{attribute 'linkalways'} 
{attribute 'no_explicit_call' := 'This FB is a CLASS and must be accessed using methods or properties'}
{attribute 'enable_dynamic_creation'}
FUNCTION_BLOCK AsyncCommand EXTENDS Disposable IMPLEMENTS I_AsyncCommand
VAR
	stateMachine : AsyncCommandStateMachine;
END_VAR

METHOD PUBLIC Abort
VAR_INPUT
END_VAR
stateMachine.Abort();
END_METHOD

PROPERTY PUBLIC Busy : BOOL
GET
IF stateMachine.IsAborted THEN
	RETURN;
END_IF

IF stateMachine.IsCompleted THEN
	RETURN;
END_IF

IF stateMachine.IsErrored THEN
	RETURN;
END_IF

IF stateMachine.IsIdle THEN
	RETURN;
END_IF

Busy := TRUE;
END_GET
END_PROPERTY

METHOD PUBLIC CyclicCall
VAR_INPUT
END_VAR
IF stateMachine.IsIdle THEN
	OnIdle();
END_IF

IF stateMachine.IsInitializing THEN
	OnInitializing(stateMachine);
END_IF

IF stateMachine.IsExecuting THEN
	OnExecuting(stateMachine);
END_IF

IF stateMachine.IsCompleting THEN
	OnCompleting(stateMachine);
END_IF

IF stateMachine.IsCompleted THEN
	OnCompleted();
END_IF

IF stateMachine.IsAborting THEN
	OnAborting(stateMachine);
END_IF

IF stateMachine.IsAborted THEN
	OnAborted();
END_IF

IF stateMachine.IsErrored THEN
	OnErrored();
END_IF
END_METHOD

PROPERTY PUBLIC Done : BOOL
GET
Done := stateMachine.IsCompleted;
END_GET
END_PROPERTY

PROPERTY PUBLIC Error : BOOL
GET
Error := stateMachine.IsErrored;
END_GET
END_PROPERTY

PROPERTY PUBLIC ErrorId : UDINT
GET
ErrorId := stateMachine.ErrorId;
END_GET
END_PROPERTY

METHOD PUBLIC Execute
VAR_INPUT
END_VAR
stateMachine.Execute();
END_METHOD

METHOD PROTECTED OnAborted
VAR_INPUT
END_VAR
END_METHOD

METHOD PROTECTED OnAborting
VAR_INPUT
	StateControl : I_AsyncCommandStateControl;
END_VAR
// default behaviour is to go to next state
// you can override this method to implement your own completing control code.
// just call StateControl.Next() when your code is completed.  

StateControl.Next();
END_METHOD

METHOD PROTECTED OnCompleted : BOOL
VAR_INPUT
END_VAR
END_METHOD

METHOD PROTECTED OnCompleting
VAR_INPUT
	StateControl : I_AsyncCommandStateControl;
END_VAR
// default behaviour is to go to next state
// you can override this method to implement your own completing control code.
// just call StateControl.Next() when your code is completed.  

StateControl.Next();
END_METHOD

METHOD PROTECTED OnErrored
VAR_INPUT
END_VAR
END_METHOD

METHOD PROTECTED OnExecuting
VAR_INPUT
	StateControl : I_AsyncCommandStateControl;
END_VAR
// default behaviour is to go to next state
// you can override this method to implement your own executing control code.
// just call StateControl.Next() when your code is completed.  

StateControl.Next();
END_METHOD

METHOD PROTECTED OnIdle
VAR_INPUT
END_VAR
END_METHOD

METHOD PROTECTED OnInitializing
VAR_INPUT
	StateControl : I_AsyncCommandStateControl;
END_VAR
// default behaviour is to go to next state
// you can override this method to implement your own initializing control code.
// just call StateControl.Next() when your code is completed.  

StateControl.Next();
END_METHOD

END_FUNCTION_BLOCK

(* stored: Version 1.1.0.1, ProductVersion 3.1.4024.12
   POU AsyncCommand: Id {c973928e-4f5b-09d1-33f2-08f2e9394838}, SpecialFunc None
   Folder Protected: Id {5a39a5d2-86a8-08f5-2eea-c36e6bea10ac}
   Method Abort: Id {7fe7ef70-8f92-07c8-094c-3e23fcd2f4b9}
   Property Busy: Id {41fde25d-7c78-0f8a-2bd6-3c43629fa217}
   Get Get: Id {50fe8db0-7c48-03a5-182b-c8bbcc843bb1}
   Method CyclicCall: Id {b75deb0d-00cc-0f69-05ee-aa8fb62f7338}
   Property Done: Id {eacbe765-c810-0ffb-3782-548f55814d64}
   Get Get: Id {37abf15d-b55d-0ce9-2e13-d50267a4f386}
   Property Error: Id {4bf62e89-ef02-06e5-150d-17a283011e29}
   Get Get: Id {1490cc77-4707-0ec6-35ed-b61401746957}
   Property ErrorId: Id {f4d11268-ec93-09a1-2668-04b067b61f26}
   Get Get: Id {98bcd037-239a-0660-2fd5-51fda5bc435f}
   Method Execute: Id {41fa219d-23fb-0366-23d6-d24f61053bbb}
   Method OnAborted: Id {7e68c239-789d-0d5c-3c67-7db5ca91e882}
   Method OnAborting: Id {08f4d610-9eda-0ffa-3e97-7ba8443c1df6}
   Method OnCompleted: Id {2c849ec3-590e-0eb7-1144-6f869779967e}
   Method OnCompleting: Id {0e9ca6ef-79ca-0dcf-0bf9-aef3ab213f65}
   Method OnErrored: Id {365e301c-f2d5-0e95-2f79-fded5f71ab0f}
   Method OnExecuting: Id {6f50fb5b-8cb8-050c-3e6b-c5c35e1efb27}
   Method OnIdle: Id {be7236a6-a37a-0c29-2b0a-0ba8ff453f72}
   Method OnInitializing: Id {491ef17d-1faf-01e9-0b5b-861a5c3ce3bc} *)
